Omron CX-Programmer project NewProject (CX-Programmer 9.41)

# PLC NewPLC1: CJ1M CPU13
I/O table (CPU CJ1M-CPU13): rack 0 slot 0 CJ1W-ETN21(ETN21Mode)

## Global symbols (name address type ; comment)
Area1_Local_UDP_TCP_port D30019 CHANNEL  ; The local UDP or TCP port number
Area1_Option_UDP_TCP_Socket D30018 CHANNEL  ; The linger and heartbeat option plus UDP or TCP socket to be opened.
Area1_Remote_IP_Address1 D30020 CHANNEL  ; The IP-address part 1 to connect to
Area1_Remote_IP_Address2 D30021 CHANNEL  ; The IP-address part 2 to connect to
Area1_Remote_UDP_TCP_port D30022 CHANNEL  ; The remote UDP or TCP number
Area1_Send_Receive_Address1 D30024 CHANNEL  ; Send or receive memory address
Area1_Send_Receive_Address2 D30025 CHANNEL  ; Send or receive memory address
Area1_Send_Receive_size D30023 CHANNEL  ; Number of bytes to send/receive
Area1_Time_Out_setting D30026 CHANNEL  ; Time out setting for UDp or TCP actions
Area1_response_code D30027 CHANNEL  ; Response code of action.
Close_request 1519.05 BOOL  ; Close Request Switch
Receive_request 1519.04 BOOL  ; Receive Request Switch
Send_request 1519.03 BOOL  ; Send Request Switch
TCP1_Number_Bytes_Received D30001 CHANNEL  ; The number of bytes that received in the TCP socket number 1.
TCP_Active_Open 1519.02 BOOL  ; TCP Active Open Request Switch
TCP_Close_Bit 0.01 BOOL  ; TCP port close request
TCP_Close_Error_FLAG 1.01 BOOL  ; There has been an error closing a TCP connection
TCP_Closing_flag 2.01 BOOL  ; The TCP port is closing.
TCP_Connection1_Status D30009 CHANNEL  ; TCP connection 1 status information
TCP_Connection2_Status D30010 CHANNEL  ; TCP connection 2 status information
TCP_Connection3_Status D30011 CHANNEL  ; TCP connection 3 status information
TCP_Connection4_Status D30012 CHANNEL  ; TCP connection 4 status information
TCP_Connection5_Status D30013 CHANNEL  ; TCP connection 5 status information
TCP_Connection6_Status D30014 CHANNEL  ; TCP connection 6 status information
TCP_Connection7_Status D30015 CHANNEL  ; TCP connection 7 status information
TCP_Connection8_Status D30016 CHANNEL  ; TCP connection 8 status information
TCP_Open_Bit 0.00 BOOL  ; Open a Passive TCP connection
TCP_Open_Error_FLAG 1.00 BOOL  ; There has been an error opening a TCP connection
TCP_Opening_Flag 2.00 BOOL  ; The Passive TCP open is processing
TCP_Passive_Open 1519.01 BOOL  ; TCP Passive Open Request Switch
TCP_Receive_Bit 0.03 BOOL  ; TCP Receive request bit
TCP_Receive_Error_Flag 1.03 BOOL  ; There has been an error receiving data
TCP_Receiving_Flag 2.03 BOOL  ; Data is being received.
TCP_Send_Bit 0.02 BOOL  ; TCP Send request bit
TCP_Send_Error_Flag 1.02 BOOL  ; There has been an error sending data
TCP_Sending_Flag 2.02 BOOL  ; Data is being sent.
TCP_Socket1_Status 1509 CHANNEL  ; Status of TCP socket number 1
TCP_Socket2_Status 1510 CHANNEL  ; Status of TCP socket number 2
TCP_Socket3_Status 1511 CHANNEL  ; Status of TCP socket number 3
TCP_Socket4_Status 1512 CHANNEL  ; Status of TCP socket number 4
TCP_Socket5_Status 1513 CHANNEL  ; Status of TCP socket number 5
TCP_Socket6_Status 1514 CHANNEL  ; Status of TCP socket number 6
TCP_Socket7_Status 1515 CHANNEL  ; Status of TCP socket number 7
TCP_Socket8_Status 1516 CHANNEL  ; Status of TCP socket number 8
UDP_Open 1519.00 BOOL  ; UDP socket opened when switch is turned ON.
UDP_Socket1_Status 1501 CHANNEL  ; Status of UDP socket number 1
UDP_Socket2_Status 1502 CHANNEL  ; Status of UDP socket number 2
UDP_Socket3_Status 1503 CHANNEL  ; Status of UDP socket number 3
UDP_Socket4_Status 1504 CHANNEL  ; Status of UDP socket number 4
UDP_Socket5_Status 1505 CHANNEL  ; Status of UDP socket number 5
UDP_Socket6_Status 1506 CHANNEL  ; Status of UDP socket number 6
UDP_Socket7_Status 1507 CHANNEL  ; Status of UDP socket number 7
UDP_Socket8_Status 1508 CHANNEL  ; Status of UDP socket number 8

## Program NewProgram1 (cyclic task 0)

### Section TCP_passive_open

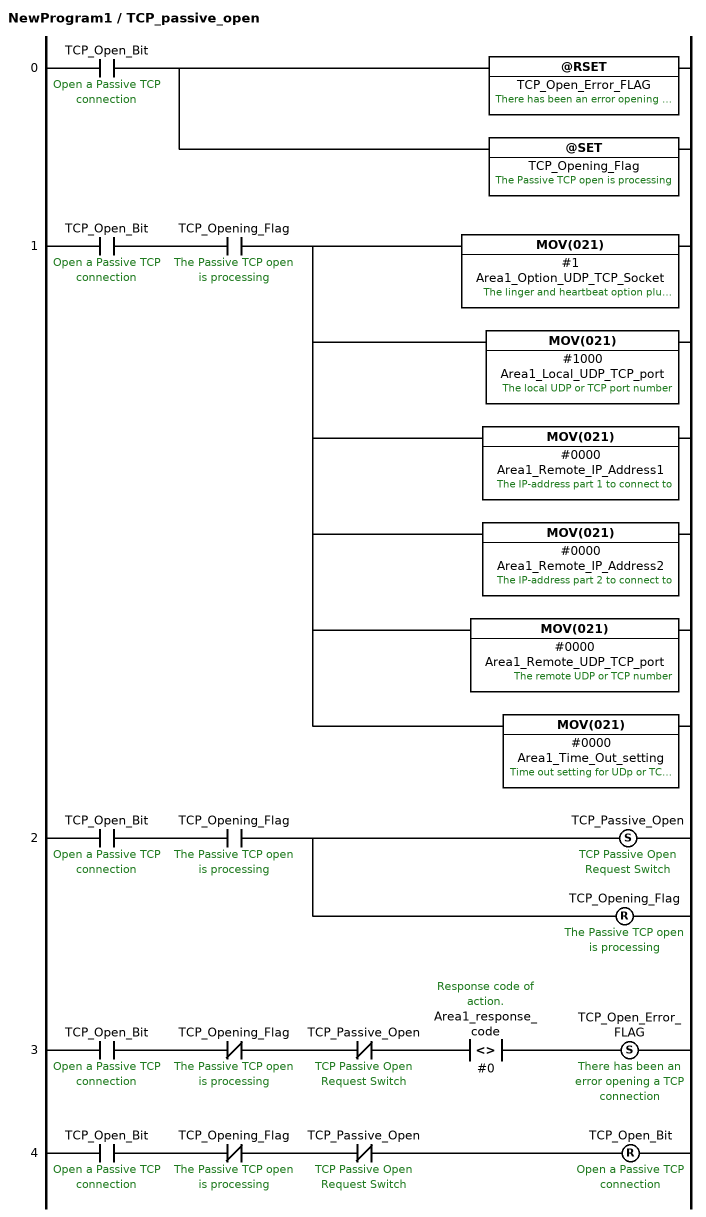
; rung 0
LD TCP_Open_Bit  ; Open a Passive TCP connection
@RSET TCP_Open_Error_FLAG  ; There has been an error opening a TCP connection
@SET TCP_Opening_Flag  ; The Passive TCP open is processing
; rung 1
LD TCP_Open_Bit  ; Open a Passive TCP connection
AND TCP_Opening_Flag  ; The Passive TCP open is processing
MOV(021) #1 Area1_Option_UDP_TCP_Socket  ; The linger and heartbeat option plus UDP or TCP socket to be opened.
MOV(021) #1000 Area1_Local_UDP_TCP_port  ; The local UDP or TCP port number
MOV(021) #0000 Area1_Remote_IP_Address1  ; The IP-address part 1 to connect to
MOV(021) #0000 Area1_Remote_IP_Address2  ; The IP-address part 2 to connect to
MOV(021) #0000 Area1_Remote_UDP_TCP_port  ; The remote UDP or TCP number
MOV(021) #0000 Area1_Time_Out_setting  ; Time out setting for UDp or TCP actions
; rung 2
LD TCP_Open_Bit  ; Open a Passive TCP connection
AND TCP_Opening_Flag  ; The Passive TCP open is processing
SET TCP_Passive_Open  ; TCP Passive Open Request Switch
RSET TCP_Opening_Flag  ; The Passive TCP open is processing
; rung 3
LD TCP_Open_Bit  ; Open a Passive TCP connection
ANDNOT TCP_Opening_Flag  ; The Passive TCP open is processing
ANDNOT TCP_Passive_Open  ; TCP Passive Open Request Switch
AND<>(305) Area1_response_code #0  ; Response code of action.
SET TCP_Open_Error_FLAG  ; There has been an error opening a TCP connection
; rung 4
LD TCP_Open_Bit  ; Open a Passive TCP connection
ANDNOT TCP_Opening_Flag  ; The Passive TCP open is processing
ANDNOT TCP_Passive_Open  ; TCP Passive Open Request Switch
RSET TCP_Open_Bit  ; Open a Passive TCP connection

### Section TCP_close

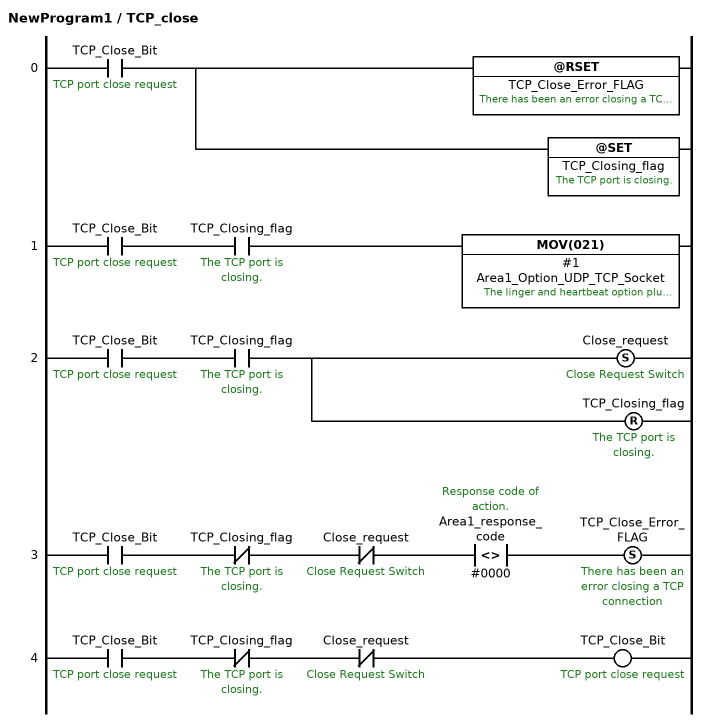
; rung 0
LD TCP_Close_Bit  ; TCP port close request
@RSET TCP_Close_Error_FLAG  ; There has been an error closing a TCP connection
@SET TCP_Closing_flag  ; The TCP port is closing.
; rung 1
LD TCP_Close_Bit  ; TCP port close request
AND TCP_Closing_flag  ; The TCP port is closing.
MOV(021) #1 Area1_Option_UDP_TCP_Socket  ; The linger and heartbeat option plus UDP or TCP socket to be opened.
; rung 2
LD TCP_Close_Bit  ; TCP port close request
AND TCP_Closing_flag  ; The TCP port is closing.
SET Close_request  ; Close Request Switch
RSET TCP_Closing_flag  ; The TCP port is closing.
; rung 3
LD TCP_Close_Bit  ; TCP port close request
ANDNOT TCP_Closing_flag  ; The TCP port is closing.
ANDNOT Close_request  ; Close Request Switch
AND<>(305) Area1_response_code #0000  ; Response code of action.
SET TCP_Close_Error_FLAG  ; There has been an error closing a TCP connection
; rung 4
LD TCP_Close_Bit  ; TCP port close request
ANDNOT TCP_Closing_flag  ; The TCP port is closing.
ANDNOT Close_request  ; Close Request Switch
OUT TCP_Close_Bit  ; TCP port close request

### Section TCP_send

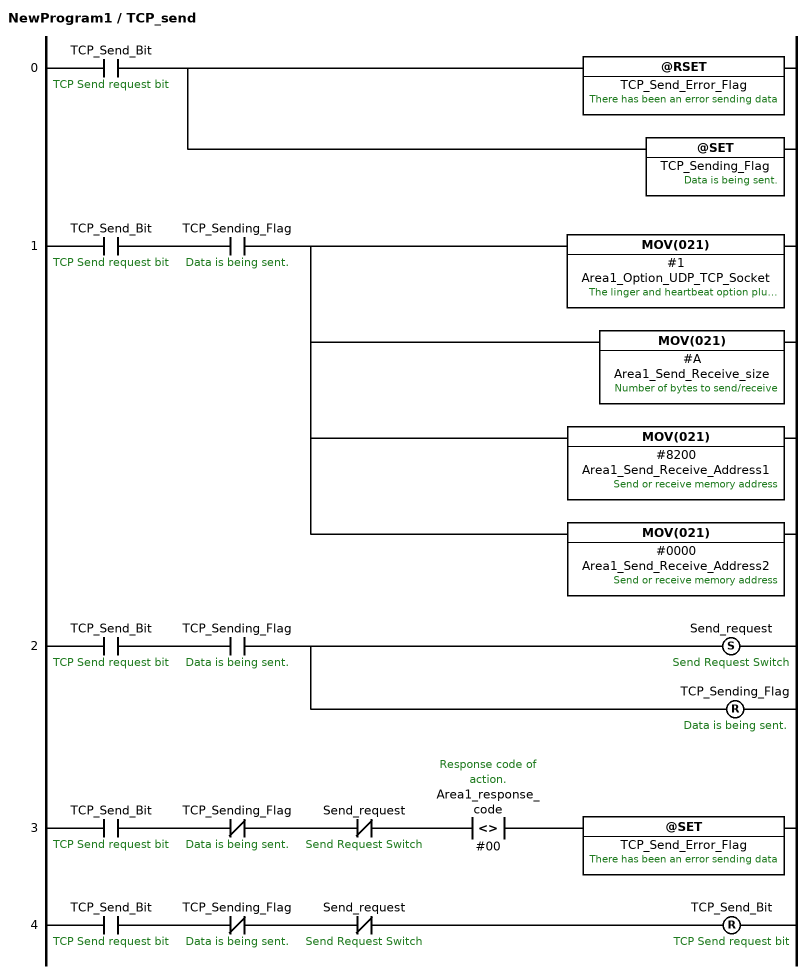
; rung 0
LD TCP_Send_Bit  ; TCP Send request bit
@RSET TCP_Send_Error_Flag  ; There has been an error sending data
@SET TCP_Sending_Flag  ; Data is being sent.
; rung 1
LD TCP_Send_Bit  ; TCP Send request bit
AND TCP_Sending_Flag  ; Data is being sent.
MOV(021) #1 Area1_Option_UDP_TCP_Socket  ; The linger and heartbeat option plus UDP or TCP socket to be opened.
MOV(021) #A Area1_Send_Receive_size  ; Number of bytes to send/receive
MOV(021) #8200 Area1_Send_Receive_Address1  ; Send or receive memory address
MOV(021) #0000 Area1_Send_Receive_Address2  ; Send or receive memory address
; rung 2
LD TCP_Send_Bit  ; TCP Send request bit
AND TCP_Sending_Flag  ; Data is being sent.
SET Send_request  ; Send Request Switch
RSET TCP_Sending_Flag  ; Data is being sent.
; rung 3
LD TCP_Send_Bit  ; TCP Send request bit
ANDNOT TCP_Sending_Flag  ; Data is being sent.
ANDNOT Send_request  ; Send Request Switch
AND<>(305) Area1_response_code #00  ; Response code of action.
@SET TCP_Send_Error_Flag  ; There has been an error sending data
; rung 4
LD TCP_Send_Bit  ; TCP Send request bit
ANDNOT TCP_Sending_Flag  ; Data is being sent.
ANDNOT Send_request  ; Send Request Switch
RSET TCP_Send_Bit  ; TCP Send request bit

### Section TCP_receive

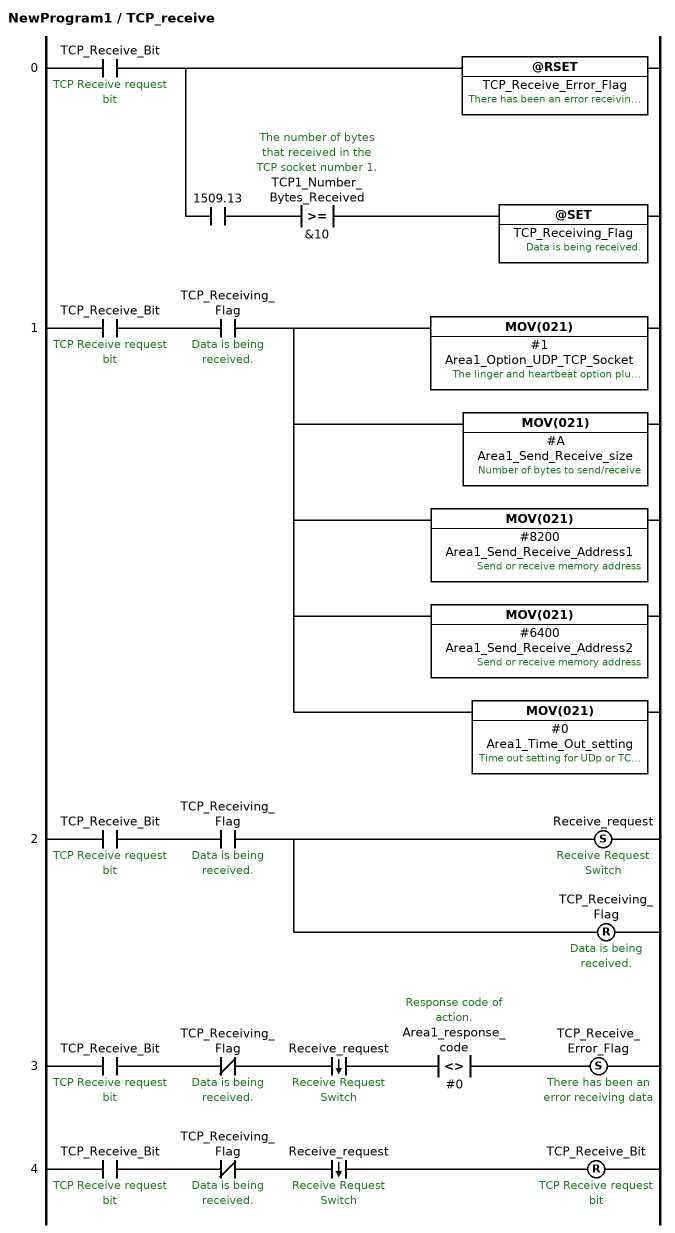
; rung 0
LD TCP_Receive_Bit  ; TCP Receive request bit
@RSET TCP_Receive_Error_Flag  ; There has been an error receiving data
AND 1509.13
AND>=(325) TCP1_Number_Bytes_Received &10  ; The number of bytes that received in the TCP socket number 1.
@SET TCP_Receiving_Flag  ; Data is being received.
; rung 1
LD TCP_Receive_Bit  ; TCP Receive request bit
AND TCP_Receiving_Flag  ; Data is being received.
MOV(021) #1 Area1_Option_UDP_TCP_Socket  ; The linger and heartbeat option plus UDP or TCP socket to be opened.
MOV(021) #A Area1_Send_Receive_size  ; Number of bytes to send/receive
MOV(021) #8200 Area1_Send_Receive_Address1  ; Send or receive memory address
MOV(021) #6400 Area1_Send_Receive_Address2  ; Send or receive memory address
MOV(021) #0 Area1_Time_Out_setting  ; Time out setting for UDp or TCP actions
; rung 2
LD TCP_Receive_Bit  ; TCP Receive request bit
AND TCP_Receiving_Flag  ; Data is being received.
SET Receive_request  ; Receive Request Switch
RSET TCP_Receiving_Flag  ; Data is being received.
; rung 3
LD TCP_Receive_Bit  ; TCP Receive request bit
ANDNOT TCP_Receiving_Flag  ; Data is being received.
%AND Receive_request  ; Receive Request Switch
AND<>(305) Area1_response_code #0  ; Response code of action.
SET TCP_Receive_Error_Flag  ; There has been an error receiving data
; rung 4
LD TCP_Receive_Bit  ; TCP Receive request bit
ANDNOT TCP_Receiving_Flag  ; Data is being received.
%AND Receive_request  ; Receive Request Switch
RSET TCP_Receive_Bit  ; TCP Receive request bit

### Section END
; rung 0
END(001)